FUNCTION_BLOCK TcUnitContext EXTENDS TcoCore.TcoContext
VAR
    _mainStation : MainStation(THIS^);

    {attribute addProperty Name "Versionsnummer Plc"}
    _sVersion : STRING(23);
    //~
    _stProgramVersion : ST_LibVersion;
    //~

END_VAR

(*~
    <docu>
        <summary>
            Main method of the TcoContext. This is the entry point of any control logic that belongs to this context.
            The call of this method is ensured by calling the <c>InstanceName.Run()</c> method, and it must not be called explicitly.
            This method is abstract, and it must be overridden in derived block.
        </summary>
    </docu>
~*)
METHOD PROTECTED Main

_mainStation();
END_METHOD

END_FUNCTION_BLOCK

(* stored: Version 1.1.0.1, ProductVersion 3.1.4024.12
   POU TcUnitContext: Id {0537339e-f15a-07ca-0b3a-11e01d7e3892}, SpecialFunc None
   Method Main: Id {9167253f-7073-00d1-1bc5-4e3d16aed3cb} *)
